(* PLC project kp15_20190419.project, CODESYS CODESYS V3.5 SP7 Patch 4 *)
(* stored: creationDateTime 2019-04-21 16:48:21.395708, modificationDateTime 2019-04-21 16:48:21.395708 *)

PROGRAM POU
  VAR
    state : INT := 0;
    i : WORD;
    j : WORD;
    res_fram_write : INT;  (* результат записи 0 - всё хорошо *)
    crc_fram_read : INT;  (* посчитанный CRC из памяти *)
    srv_104 : RLTNU.IEC104Server ;  (* IEC 104 *)
    db_104 : RLTNU.IECDB ;
    ts_104 : ARRAY[1..q_ts_full] OF RLTNU.IEC_M_SP_NA ;  (* мой массив бит на передачу в 104 *)
    tf_104 : ARRAY[1..(2 * q_ti_full)] OF RLTNU.IEC_M_ME_NC ;  (* мой массив float на передачу в 104 *)
    tu_104 : ARRAY[1..q_tu_full] OF RLTNU.IECCommand ;  (* массив команд в 104 *)
    trf_104 : ARRAY[1..q_tr_full] OF RLTNU.IECCommand ;  (* массив ТР в 104 *)
    cmd_104 : RLTNU.IECCommand ;
    event : RLTNU.IECSpontaneousEvent ;
    sys_tick : CAA.TICK ;  (* Время *)
    sys_tick_bool : BOOL;
    current_time : UDINT;
    hiTime : ULINT;
    Start_timer : TON;  (* Таймер первого запуска *)
    First_start : BOOL;  (* Флаг первого запуска *)
  END_VAR

END_PROGRAM
